Yaskawa INFORM job: R2_W28-29-A2(90,-90)_MP_OK.JBI

/JOB
//NAME R2_W28-29-A2(90,-90)_MP_OK
///FOLDERNAME MP_TEST
//POS
///NPOS 91,91,0,2,0,0
///TOOL 0
///POSTYPE PULSE
///PULSE
C00000=134097,35363,-2629,-3509,85687,4195
C00001=134100,35319,-2657,-3509,85682,4196
C00002=134101,35301,-2668,-3510,85679,4196
C00003=134097,35299,-2647,-3509,85666,4195
C00004=134099,35283,-2663,-3509,85667,4196
C00005=134097,35299,-2647,-3509,85666,4195
C00006=134101,35301,-2668,-3510,85679,4196
C00007=134110,35180,-2769,-3512,85680,4199
C00008=134109,35180,-2762,-3512,85676,4199
C00009=134110,35180,-2769,-3512,85680,4199
C00010=134101,35301,-2668,-3510,85679,4196
C00011=134097,35393,-2601,-3509,85685,4195
C00012=134098,35347,-2619,-3509,85673,4196
C00013=134099,35336,-2626,-3509,85672,4196
C00014=134098,35347,-2619,-3509,85673,4196
C00015=134097,35393,-2601,-3509,85685,4195
C00016=134101,35301,-2668,-3510,85679,4196
C00017=134100,35319,-2657,-3509,85682,4196
C00018=134097,35363,-2629,-3509,85687,4195
C00019=134087,15629,7013,-29258,40313,-40546
C00020=134115,22264,30229,-37616,31138,-35946
C00021=134121,24068,34875,-39678,29613,-34876
C00022=127111,-29209,-4000,-6420,15771,-47301
C00023=133695,22776,34807,-40008,28936,-34735
C00024=134118,23971,34630,-39562,29690,-34936
C00025=123627,-24951,-1125,1954,16097,-51447
C00026=120666,-20528,1995,8690,16640,-54794
C00027=134126,24072,34933,-39720,29589,-34854
C00028=134120,22264,30283,-37653,31113,-35926
C00029=134092,15611,7047,-29279,40288,-40534
C00030=134080,15733,6890,-49816,57800,-27924
C00031=134108,22291,30027,-55958,51058,-23118
C00032=134114,24079,34667,-57281,49961,-22172
C00033=134117,24976,36885,-57921,49462,-21720
C00034=134082,22461,34284,-57695,49610,-21883
C00035=134111,23983,34427,-57211,50014,-22221
C00036=134118,25021,37012,-57963,49430,-21691
C00037=134119,24949,36859,-57924,49462,-21719
C00038=133963,24955,36887,-57898,49361,-21751
C00039=134118,24078,34731,-57309,49941,-22152
C00040=134112,22286,30086,-55985,51038,-23098
C00041=134083,15706,6926,-49834,57778,-27909
C00042=107314,15986,7579,30647,40548,40199
C00043=107347,22706,30901,39206,31481,35470
C00044=107354,24529,35583,41313,29974,34374
C00045=107366,25500,37751,42281,29337,33877
C00046=107351,24434,35343,41203,30051,34431
C00047=107778,23220,35488,41668,29309,34219
C00048=107358,25372,37632,42277,29350,33879
C00049=107360,25386,37643,42278,29347,33881
C00050=107361,25413,37697,42298,29331,33867
C00051=107358,24533,35545,41280,29992,34391
C00052=107352,22713,30866,39176,31499,35486
C00053=107318,16007,7558,30629,40567,40209
C00054=107307,15886,7711,50986,58027,27606
C00055=107341,22685,31115,57162,51399,22737
C00056=107348,24525,35806,58487,50324,21784
C00057=107354,25474,38067,59125,49837,21332
C00058=107345,24429,35561,58416,50381,21834
C00059=107377,22914,35421,58899,49988,21495
C00060=107334,25150,37698,59089,49876,21356
C00061=107337,25169,37693,59080,49883,21363
C00062=107334,25012,37445,59027,49927,21400
C00063=107351,24527,35748,58460,50342,21804
C00064=107344,22691,31062,57137,51418,22756
C00065=107311,15912,7678,50969,58047,27621
C00066=107224,98231,89024,-42145,91889,-79190
C00067=107226,114154,117962,-42140,84639,-76250
C00068=107227,113558,117124,-42131,84797,-76314
C00069=107228,114314,118312,-42145,84539,-76209
C00070=107224,107909,108045,-42052,86817,-77135
C00071=107469,120694,126678,-42206,83245,-75576
C00072=107226,113670,117355,-42136,84735,-76290
C00073=107220,113095,116584,-42129,84867,-76346
C00074=106962,103969,104202,-42547,85649,-77974
C00075=107218,112797,116120,-42123,84964,-76386
C00076=107217,113333,116872,-42130,84823,-76329
C00077=107215,98053,88903,-42145,91872,-79188
C00078=107191,97022,87713,38294,104991,71848
C00079=107193,110152,112571,36998,98139,69405
C00080=107196,109935,112255,37008,98205,69429
C00081=107197,111121,114167,36948,97746,69272
C00082=107179,120555,126678,36679,95446,68481
C00083=107193,105706,105176,37271,99966,70039
C00084=107198,110911,113805,36959,97842,69305
C00085=107193,111229,114383,36937,97688,69250
C00086=107486,109117,111360,37102,98188,69544
C00087=107200,110699,113300,36982,98001,69361
C00088=107197,110935,113641,36971,97931,69335
C00089=107195,97212,87856,38297,104997,71852
C00090=107469,103937,96490,38021,103397,71385
BC00000=261732,528229,920609
BC00001=261667,522771,901696
BC00002=261641,520587,894131
BC00003=260063,513635,894282
BC00004=260050,513623,886217
BC00005=260063,513635,894282
BC00006=261641,520587,894131
BC00007=276947,517313,870059
BC00008=276436,515063,870108
BC00009=276947,517313,870059
BC00010=261641,520587,894131
BC00011=241964,524742,894419
BC00012=239846,515537,872576
BC00013=242180,515044,872542
BC00014=239846,515537,872576
BC00015=241964,524742,894419
BC00016=261641,520587,894131
BC00017=261667,522771,901696
BC00018=261732,528229,920609
BC00019=261754,541910,1075175
BC00020=261631,541942,1075175
BC00021=260317,536344,1075175
BC00022=259791,479805,1075175
BC00023=259791,534105,1075175
BC00024=259791,534105,1075175
BC00025=259791,479805,1075175
BC00026=259791,479805,1075175
BC00027=273200,526000,1075175
BC00028=274514,531597,1075175
BC00029=274637,531566,1075175
BC00030=199183,529416,1075175
BC00031=199060,529448,1075175
BC00032=200581,523909,1075175
BC00033=201189,521694,1075175
BC00034=201189,521694,1075175
BC00035=201189,521694,1075175
BC00036=205860,520722,1075175
BC00037=213287,519170,1075175
BC00038=217956,518191,1075175
BC00039=217348,520406,1075175
BC00040=215827,525944,1075175
BC00041=215950,525913,1075175
BC00042=175809,542354,1075175
BC00043=175686,542386,1075175
BC00044=176913,536779,1075175
BC00045=177404,534536,1075175
BC00046=177404,534536,1075175
BC00047=177404,534536,1075175
BC00048=173711,531613,1075175
BC00049=168136,527208,1075175
BC00050=164438,524289,1075175
BC00051=163947,526532,1075175
BC00052=162719,532139,1075175
BC00053=162842,532107,1075175
BC00054=238508,529497,1075175
BC00055=238385,529529,1075175
BC00056=236779,524002,1075175
BC00057=236136,521791,1075175
BC00058=236136,521791,1075175
BC00059=236136,521791,1075175
BC00060=231458,520854,1075175
BC00061=224018,519359,1075175
BC00062=219342,518414,1075175
BC00063=219984,520625,1075175
BC00064=221590,526152,1075175
BC00065=221713,526120,1075175
BC00066=93870,467997,1075175
BC00067=93820,467811,1013826
BC00068=97584,472208,995815
BC00069=99090,473967,988610
BC00070=99090,473967,988610
BC00071=99090,473967,988610
BC00072=103756,472976,988532
BC00073=123757,468753,988239
BC00074=128426,467772,988180
BC00075=126920,466013,995385
BC00076=123156,461616,1013396
BC00077=123207,461803,1075175
BC00078=241618,467265,1075175
BC00079=241568,467079,1012856
BC00080=237802,471520,994982
BC00081=236296,473297,987833
BC00082=236296,473297,987833
BC00083=236296,473297,987833
BC00084=231617,472361,987925
BC00085=211565,468374,988363
BC00086=206884,467448,988475
BC00087=208390,465671,995625
BC00088=212156,461230,1013499
BC00089=212206,461416,1075175
///LIMIT ON
BC00090=212206,759690,1075175
///POSTYPE BASE
///LIMIT OFF
///RECTAN
///RCONF 0,0,0,0,1,0,0,0,0,0,0,0,0,0,0,0,0,0,0,0,0,0,0,0
P00006=2.006,1.622,-0.565,0.0000,0.0000,0.0000
P00022=2.006,1.622,-0.565,0.0000,0.0000,0.0000
//INST
///DATE 2023/12/01 10:31
///ATTR SC,RW
///GROUP1 RB1,BS1
NOP
'r2_W28-29-A2(90,-90)
'Path S859
SFTOF
MOVL C00000 BC00000 V=1000.0
MOVL C00001 BC00001 V=400.0
MOVL C00002 BC00002 V=100.0
MOVL C00003 BC00003 V=60.0
REFP 3 C00004 BC00004
CALL JOB:SEARCH-R1
SET P022 P006
SFTON P022
MOVL C00005 BC00005 V=60.0
MOVL C00006 BC00006 V=100.0
MOVL C00007 BC00007 V=60.0
REFP 3 C00008 BC00008
CALL JOB:SEARCH-R1
SET P022 P006
SFTON P022
MOVL C00009 BC00009 V=60.0
MOVL C00010 BC00010 V=100.0
MOVL C00011 BC00011 V=100.0
MOVL C00012 BC00012 V=60.0
REFP 3 C00013 BC00013
CALL JOB:SEARCH-R1
SET P022 P006
SFTON P022
MOVL C00014 BC00014 V=60.0
MOVL C00015 BC00015 V=100.0
MOVL C00016 BC00016 V=100.0
MOVL C00017 BC00017 V=400.0
MOVL C00018 BC00018 V=1000.0
'Path W860
SFTOF
SFTON P022
MOVJ C00019 BC00019 VJ=100.00
MOVL C00020 BC00020 V=1000.0
MOVL C00021 BC00021 V=400.0
MOVL C00022 BC00022 V=100.0 PL=0
REFP 1 C00023 BC00023
REFP 2 C00024 BC00024
MACRO1 MJ#(0) ARGF6
ARCON
MOVL C00025 BC00025 V=8.3
MOVL C00026 BC00026 V=8.3
ARCOF
MOVL C00027 BC00027 V=400.0
MOVL C00028 BC00028 V=1000.0
MOVL C00029 BC00029 V=1000.0
SFTOF
'Path W861
SFTOF
SFTON P022
MOVJ C00030 BC00030 VJ=100.00
MOVL C00031 BC00031 V=1000.0
MOVL C00032 BC00032 V=400.0
MOVL C00033 BC00033 V=100.0 PL=0
REFP 1 C00034 BC00034
REFP 2 C00035 BC00035
MACRO1 MJ#(0) ARGF6
ARCON
MOVL C00036 BC00036 V=8.3
MOVL C00037 BC00037 V=8.3
MOVL C00038 BC00038 V=8.3
ARCOF
MOVL C00039 BC00039 V=400.0
MOVL C00040 BC00040 V=1000.0
MOVL C00041 BC00041 V=1000.0
SFTOF
'Path W862
SFTOF
SFTON P022
MOVJ C00042 BC00042 VJ=100.00
MOVL C00043 BC00043 V=1000.0
MOVL C00044 BC00044 V=400.0
MOVL C00045 BC00045 V=100.0 PL=0
REFP 1 C00046 BC00046
REFP 2 C00047 BC00047
MACRO1 MJ#(0) ARGF6
ARCON
MOVL C00048 BC00048 V=8.3
MOVL C00049 BC00049 V=8.3
MOVL C00050 BC00050 V=8.3
ARCOF
MOVL C00051 BC00051 V=400.0
MOVL C00052 BC00052 V=1000.0
MOVL C00053 BC00053 V=1000.0
SFTOF
'Path W863
SFTOF
SFTON P022
MOVJ C00054 BC00054 VJ=100.00
MOVL C00055 BC00055 V=1000.0
MOVL C00056 BC00056 V=400.0
MOVL C00057 BC00057 V=100.0 PL=0
REFP 1 C00058 BC00058
REFP 2 C00059 BC00059
MACRO1 MJ#(0) ARGF6
ARCON
MOVL C00060 BC00060 V=8.3
MOVL C00061 BC00061 V=8.3
MOVL C00062 BC00062 V=8.3
ARCOF
MOVL C00063 BC00063 V=400.0
MOVL C00064 BC00064 V=1000.0
MOVL C00065 BC00065 V=1000.0
SFTOF
'
'Path W864
SFTOF
SFTON P022
MOVJ C00066 BC00066 VJ=100.00
MOVL C00067 BC00067 V=1000.0
MOVL C00068 BC00068 V=400.0
MOVL C00069 BC00069 V=100.0 PL=0
REFP 1 C00070 BC00070
REFP 2 C00071 BC00071
MACRO1 MJ#(0) ARGF6
ARCON
MOVL C00072 BC00072 V=8.3
MOVL C00073 BC00073 V=8.3
MOVL C00074 BC00074 V=8.3
ARCOF
MOVL C00075 BC00075 V=400.0
MOVL C00076 BC00076 V=1000.0
MOVL C00077 BC00077 V=1000.0
SFTOF
'Path W865
SFTOF
SFTON P022
MOVJ C00078 BC00078 VJ=100.00
MOVL C00079 BC00079 V=1000.0
MOVL C00080 BC00080 V=400.0
MOVL C00081 BC00081 V=100.0 PL=0
REFP 1 C00082 BC00082
REFP 2 C00083 BC00083
MACRO1 MJ#(0) ARGF6
ARCON
MOVL C00084 BC00084 V=8.3
MOVL C00085 BC00085 V=8.3
MOVL C00086 BC00086 V=8.3
ARCOF
MOVL C00087 BC00087 V=400.0
MOVL C00088 BC00088 V=1000.0
MOVL C00089 BC00089 V=1000.0
SFTOF
MOVJ C00090 BC00090 VJ=100.00
END
